{attribute 'GeneratedUsingTerminal: EP1518-0002-0016'}
{attribute addProperty BoxType "EP1518-0002-0016"}
{attribute addProperty Id "InputAT %I*ARRAY[0..7] OF BOOL8"}
{attribute addProperty CRC "3697175534"}
{attribute addProperty Size "8"}
TYPE DIG_Inputs_CAFF6004 EXTENDS InputBase_8311D824 :
STRUCT
	{attribute addProperty Name "Input"}
	Input AT %I* : ARRAY[0..7] OF BOOL;
END_STRUCT
END_TYPE

(* stored: Version 1.2.0.0, ProductVersion 3.1.4024.11
   DUT DIG_Inputs_CAFF6004: Id {8c01efa8-4423-4d36-8d3c-d4756ef60111} *)
